FUNCTION_BLOCK EA_LeftPublishSubscribeAdapter_0
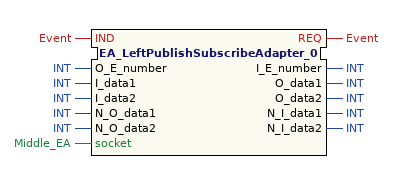
  EVENT_INPUT
    IND;
  END_EVENT
  EVENT_OUTPUT
    REQ;
  END_EVENT
  VAR_INPUT
    O_E_number : INT;
    I_data1 : INT;
    I_data2 : INT;
    N_O_data1 : INT;
    N_O_data2 : INT;
  END_VAR
  VAR_OUTPUT
    I_E_number : INT;
    O_data1 : INT;
    O_data2 : INT;
    N_I_data1 : INT;
    N_I_data2 : INT;
  END_VAR
  SOCKETS
    socket : Middle_EA;
  END_SOCKETS
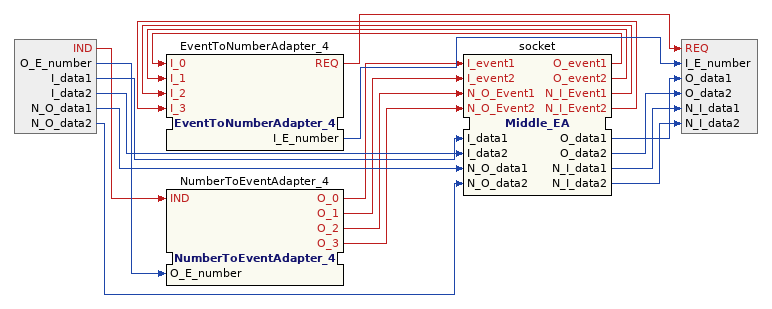
  FBS
    EventToNumberAdapter_4 : EventToNumberAdapter_4;
    NumberToEventAdapter_4 : NumberToEventAdapter_4;
  END_FBS
  EVENT_CONNECTIONS
    IND TO NumberToEventAdapter_4.IND;
    NumberToEventAdapter_4.O_0 TO socket.I_event1;
    NumberToEventAdapter_4.O_1 TO socket.I_event2;
    NumberToEventAdapter_4.O_2 TO socket.N_O_Event1;
    NumberToEventAdapter_4.O_3 TO socket.N_O_Event2;
    socket.O_event1 TO EventToNumberAdapter_4.I_0;
    socket.O_event2 TO EventToNumberAdapter_4.I_1;
    socket.N_I_Event1 TO EventToNumberAdapter_4.I_2;
    socket.N_I_Event2 TO EventToNumberAdapter_4.I_3;
    EventToNumberAdapter_4.REQ TO REQ;
  END_CONNECTIONS
  DATA_CONNECTIONS
    O_E_number TO NumberToEventAdapter_4.O_E_number;
    EventToNumberAdapter_4.I_E_number TO I_E_number;
    I_data1 TO socket.I_data1;
    I_data2 TO socket.I_data2;
    N_O_data1 TO socket.N_O_data1;
    N_O_data2 TO socket.N_O_data2;
    socket.O_data1 TO O_data1;
    socket.O_data2 TO O_data2;
    socket.N_I_data1 TO N_I_data1;
    socket.N_I_data2 TO N_I_data2;
  END_CONNECTIONS
END_FUNCTION_BLOCK
